TYPE T_PCM_Filename : T_MaxString;
END_TYPE

(* stored: Version 1.1.0.1, ProductVersion 3.1.4024.15
   DUT T_PCM_Filename: Id {68bacc27-ddb5-44d0-8203-ead204928a4a} *)
